FUNCTION HYST_2 (* Hystereses function *)
  (* Standard: 61499-1 *)
  (* Version 1.0, 2025-12-21, franz *)
  PACKAGE OSCAT::Basic::POUs::Engineering::Control;
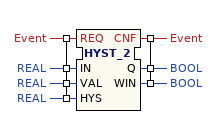
  EVENT_INPUT
    REQ WITH IN, VAL, HYS;
  END_EVENT
  EVENT_OUTPUT
    CNF WITH Q, WIN;
  END_EVENT
  VAR_INPUT
    IN : REAL;
    VAL : REAL;
    HYS : REAL;
  END_VAR
  VAR_OUTPUT
    Q : BOOL;
    WIN : BOOL;
  END_VAR
  BODY IN ST:
PACKAGE OSCAT::Basic::POUs::Engineering::Control;

(* Hystereses function *)
FUNCTION HYST_2
VAR_INPUT
	IN : REAL;
	VAL : REAL;
	HYS : REAL;
END_VAR
VAR_OUTPUT
	Q : BOOL;
	WIN : BOOL;
END_VAR
VAR
	tmp : REAL;
END_VAR

(*
 * version 1.2	2. jun. 2008 programmer 	oscat tested BY	oscat
 * *
 * this hysteresis function switches the output high if the input signal reaches obove val + hys/2
 * and will switch to low when the input falls back below val - hys/2 value.
 * a separate output mid is set if the input stays between low and high value.
 *)
tmp := VAL - HYS * 0.5;
IF IN < tmp THEN
	Q := FALSE;
	WIN := FALSE;
ELSIF IN > tmp + HYS THEN
	Q := TRUE;
	WIN := FALSE;
ELSE
	WIN := TRUE;
END_IF;

END_FUNCTION

(* revision history hm		4. aug 2006	rev 1.0 original version
 *
 * hm		5. jan 2008	rev 1.1 improved code for better performance
 *
 * hm		2. jun. 2008	rev 1.2 improved performance *)
  END_BODY
END_FUNCTION
